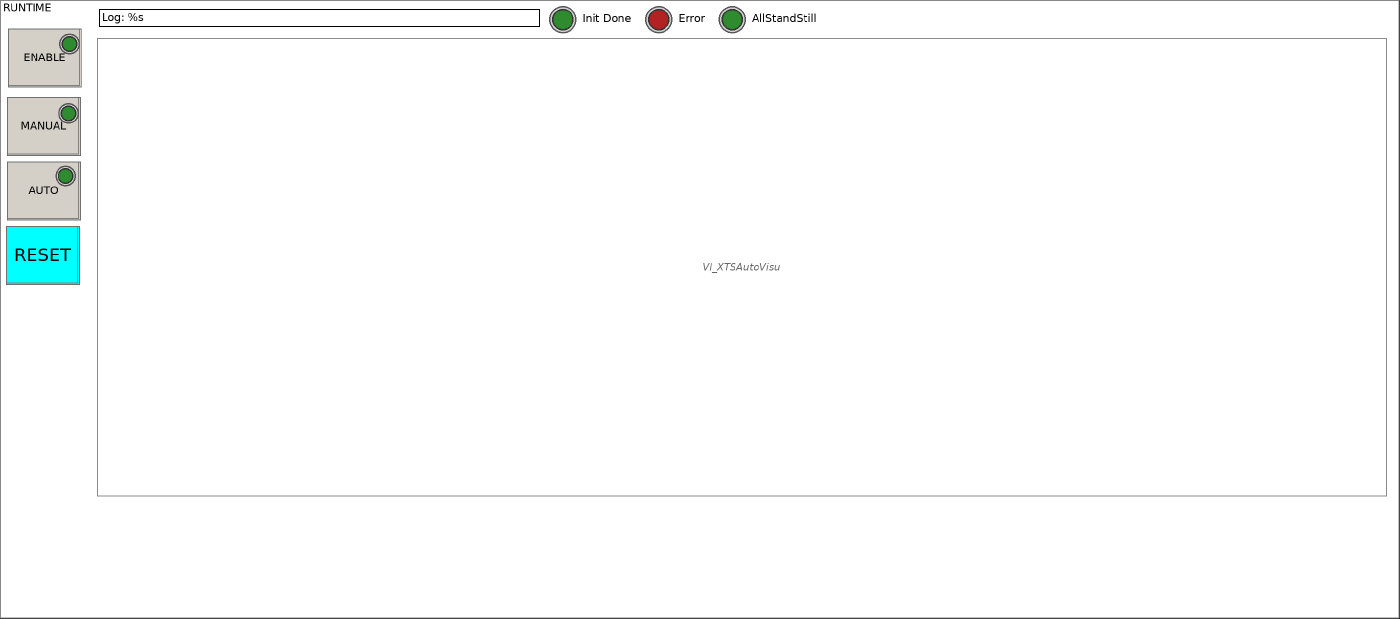
VISUALIZATION VI_XTSRunTimeVisu  // 1430x633
VAR_IN_OUT
	xts : XTS_System;
END_VAR
    Rectangle (0,0 1430x633), "RUNTIME"
    Button (8,29 75x60), "ENABLE"
        toggle xts.bEnable
    Button (7,99 75x60), "MANUAL", input disabled if: xts.bInAutomatic = TRUE
        toggle xts.bManual
        OnMouseClick: FrameSelectionChange Selection=SelectedFrame=a18850ea-e303-4efa-b84e-5057b211b999, Selection=1, GlobSel=AssignType=Directly, SelType=Locally
    Button (7,165 75x60), "AUTO", input disabled if: xts.bInManual = TRUE
        toggle xts.bAutomatic
        OnMouseClick: FrameSelectionChange Selection=SelectedFrame=a18850ea-e303-4efa-b84e-5057b211b999, GlobSel=AssignType=Directly, SelType=Locally
    Lamp1 (559,4 32x32), variable: xts.bInitDone, style: Lamp-Lamp1-Green
    Label (592,4 110x30), "Init Done"
    Lamp1 (657,4 32x32), variable: xts.bError, style: Lamp-Lamp1-Red
    Label (690,4 110x30), "Error"
    Lamp1 (732,4 32x32), variable: xts.bAllMoversStandStill, style: Lamp-Lamp1-Green
    Label (765,4 110x30), "AllStandStill"
    Lamp1 (59,32 24x26), variable: xts.bEnabled, style: Lamp-Lamp1-Green
    Rectangle (101,9 450x18), "Log: %s", text variable: xts.sLog
        OnMouseClick: write the text variable via Default
    Frame (99,39 1317x468)
        shows VI_XTSAutoVisu(xts := xts)
        shows VI_XTSManualVisu(xts := xts)
    Lamp1 (55,167 24x26), variable: xts.bInAutomatic=true, style: Lamp-Lamp1-Green
    Lamp1 (58,103 24x26), variable: xts.bInManual=true, style: Lamp-Lamp1-Green
    Button (6,231 75x60), "RESET"
        tap xts.bReset
END_VISUALIZATION

(* stored: Version 1.1.0.1, ProductVersion 3.1.4024.11
   Visu VI_XTSRunTimeVisu: Id {7519b7d6-9bdb-4064-9291-04f668dd61c0} *)
